FUNCTION_BLOCK Environment
VAR_INPUT
END_VAR
VAR_OUTPUT
	
MaxTableYTravel 		: LREAL ; 
MaxTableXTravel 		: LREAL ;
		             
MinTableYTravel 		: LREAL ; 
MinTableXTravel 		: LREAL ; 

END_VAR
VAR
END_VAR

METHOD Boundry 
VAR_INPUT
	
			NumberOfXTiles				: INT;
			NumberOfYTiles				: INT; 
			MoverTypeWidth 				: LREAL;
		    MoverTypeLength				: LREAL;
			
END_VAR 

VAR 
			Buffer						: INT := 5; 
END_VAR
MaxTableYTravel := (NumberOfYTiles * 240) - MoverTypeWidth  - Buffer;
MaxTableXTravel := (NumberOfXTiles * 240) - MoverTypeLength - Buffer;
		
MinTableYTravel :=  MoverTypeWidth   + Buffer;
MinTableXTravel :=  MoverTypeLength  + Buffer;
END_METHOD

METHOD Forces 
VAR_INPUT
END_VAR
END_METHOD

END_FUNCTION_BLOCK

(* stored: Version 1.1.0.1, ProductVersion 3.1.4024.12
   POU Environment: Id {bc804a70-ba27-434f-a722-0a692fdcb6d7}, SpecialFunc None
   Method Boundry: Id {bdc5a1ba-4bdc-4f6e-891d-211745460f60}
   Method Forces: Id {97bf2863-1c46-48a8-8c41-067ed868cafd} *)
